TYPE ST_StationParams :
STRUCT
	fMinX		: LREAL;
	fMaxX		: LREAL;
	fMinY		: LREAL;
	fMaxY		: LREAL;
END_STRUCT
END_TYPE

(* stored: Version 1.1.0.1
   DUT ST_StationParams: Id {385c7f81-cc01-4a04-b8c8-6b7de3aa0cb8} *)
